{region '#Template'}
	{attribute 'Version' := '1.2.1.0'}
	{attribute 'Tags' := '"LCID": "1031", "Text": "General, Settings, Project, Basics"'}
	{attribute 'Tags' := '"LCID": "1033", "Text": "General, Settings, Project, Basics"'}
	{attribute 'Description' := '"LCID": "1031", "Text": "Basis Einstellungen der Steuerung, system services"'}
	{attribute 'Description' := '"LCID": "1033", "Text": "Basic settings of the control"'}
{endregion}
FUNCTION_BLOCK FB_BA_IFP EXTENDS FB_BA_View
VAR_INPUT
END_VAR
VAR_INPUT CONSTANT
	Trend				: FB_BA_TrendLogging;	
	Project				: FB_BA_ProjectEx;
END_VAR
VAR_OUTPUT
END_VAR
VAR
	LblProject			: FB_BA_Label2x :=(iAggregate:=LblAggregates_AutomationStationEquipment,	 iFunction:=LblControl_BACnetDevice);
END_VAR

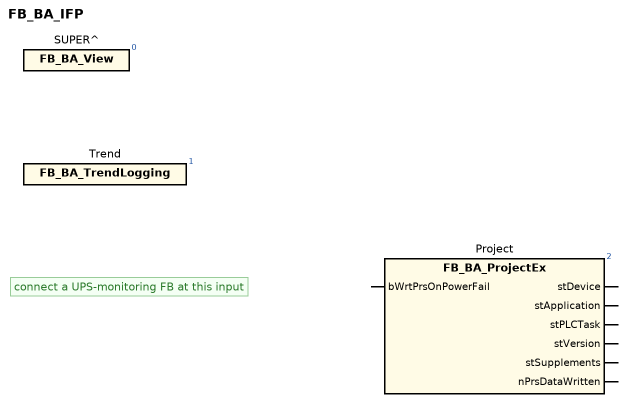
SUPER^(); // FB_BA_View
Trend(); // FB_BA_TrendLogging
// connect a UPS-monitoring FB at this input
Project(); // FB_BA_ProjectEx

METHOD FB_init : BOOL
VAR_INPUT
	bInitRetains : BOOL; // if TRUE, the retain variables are initialized (warm start / cold start)
	bInCopyCode : BOOL;  // if TRUE, the instance afterwards gets moved into the copy code (online change)
END_VAR
Project.iParent						:= THIS^;
Project.iLabel						:= LblProject;

Project.tPrsData_DefaultPeriod 		:= T#30M;
Project.tPrsData_ComissioningPeriod := T#10M;

Trend.iParent						:= THIS^;
Trend.iLabel						:= LblControl_TrendLogging;
Trend.sObjectName					:= '{Idx=01}';
Trend.eDPADMode						:= E_BA_DPADMode.eInclude;
END_METHOD

END_FUNCTION_BLOCK

(* stored: Version 1.1.0.1, ProductVersion 3.1.4024.9
   POU FB_BA_IFP: Id {783a29aa-bcf7-4dde-82ff-593bf793d1e3}, SpecialFunc None
   Method FB_init: Id {a6ea51b1-fc25-4891-bcad-ddbebe33c60e} *)
